{attribute 'GeneratedUsingTerminal: EK1122-0000-0018'}
{attribute addProperty BoxType "EK1122-0000-0018"}
{attribute addProperty Id "Beckhoff_EL25xxsub_EK1100EK1100_1FC0878B2"}
{attribute addProperty CRC "2201281511"}
{attribute addProperty Size "2"}
TYPE Beckhoff_EL25xxEK1122_8334E3E7 EXTENDS EK1122_1FC0878B :
STRUCT
	{attribute addProperty Name "Beckhoff_EL25xxsub_EK1100"}
	{attribute addProperty PreviousPort "Beckhoff EL25xxEK1122 : D"}
	Beckhoff_EL25xxsub_EK1100 : EK1100_1FC0878B;
END_STRUCT
END_TYPE

(* stored: Version 1.2.0.0, ProductVersion 3.1.4024.9
   DUT Beckhoff_EL25xxEK1122_8334E3E7: Id {bbb20a5a-c95f-4cfb-b1a3-092b2d2bd2a7} *)
